// Sequential SDOs at startup or when forced; parallel writes otherwise (mirrors Homing Params block).
FUNCTION_BLOCK FB_WriteStepModeParameters
VAR_INPUT
    bEnable : BOOL;
END_VAR
VAR_IN_OUT
    stDS402Drive         : ST_DS402Drive;
    stMotionStage        : ST_MotionStage;
    stMCS2ChanParameter	: ST_MCS2ChanParameter;
END_VAR

VAR_OUTPUT
   bStepModeParamsSet : BOOL;
END_VAR
VAR
    // ====== Measurements & scaled values ======
    {attribute 'hide'}
    nScaledFErrWin          : DINT;
    {attribute 'hide'}
    nScalededSteps          : DINT;
    {attribute 'hide'}
    fScalededSteps          : LREAL;
    {attribute 'hide'}
    fMeasuredVelo           : LREAL;
    {attribute 'hide'}
    fMeasuredAcc            : LREAL;
    {attribute 'hide'}
    fParameterValue         : LREAL;
    {attribute 'hide'}
    fMeasuredPos             : LREAL;
    // ====== Internal numeric parameters ======
    {attribute 'hide'}
    nScalededStepAmp         : UINT;
    {attribute 'hide'}
    nScaledStepFreq          : UINT;
    // Open Loop Operations
    {attribute 'hide'}
    fbSetSteps          : FB_EcCoESdoWrite;
    {attribute 'hide'}
    fbSetStepFreq       : FB_EcCoESdoWrite;
    {attribute 'hide'}
    fbSetStepAmp        : FB_EcCoESdoWrite;
    {attribute 'hide'}
    nRecentSteps        : DINT;
    {attribute 'hide'}
    nRecentStepAmp      : UINT;
    {attribute 'hide'}
    nRecentStepFreq     : UINT;
    {attribute 'hide'}
    ftStepAmpUpdateDone : F_TRIG;
    {attribute 'hide'}
    ftStepFreqUpdateDone    : F_TRIG;
    {attribute 'hide'}
    ftStepUpdateDone    : F_TRIG;
    tonStartUp : TON;
    nJogParamStep : INT := 0; // 0=idle/start, 1=steps, 2=amp, 3=freq, 10=done, -1=error
    bForceSequentialSDOs : BOOL := FALSE;
    bErrorAcknowledge: BOOL;
END_VAR

IF bEnable THEN
    tonStartUp(
        IN := bEnable AND NOT bStepModeParamsSet,
        PT := T#4S
    );
    IF (NOT tonStartUp.Q) AND (nJogParamStep <> 0) AND (NOT bForceSequentialSDOs) THEN
        nJogParamStep := 0;
    END_IF

    IF (nJogParamStep = -1) AND bErrorAcknowledge THEN
        nJogParamStep := 0;
        stMotionStage.bError := FALSE;
        stMotionStage.nErrorId := 0;
    END_IF
    ScaleStepModeParams();

    ftStepUpdateDone   (CLK := fbSetSteps.bBusy);
    ftStepAmpUpdateDone(CLK := fbSetStepAmp.bBusy);
    ftStepFreqUpdateDone(CLK := fbSetStepFreq.bBusy);

    IF tonStartUp.Q OR bForceSequentialSDOs THEN
        CASE nJogParamStep OF
        0:
            bStepModeParamsSet := FALSE;
            fbSetSteps.bExecute     := FALSE;
            fbSetStepAmp.bExecute   := FALSE;
            fbSetStepFreq.bExecute  := FALSE;
            nJogParamStep := 1;

        1: // Set Steps
            IF (nScalededSteps <> nRecentSteps) THEN
                fbSetSteps.bExecute := TRUE;
                IF ftStepUpdateDone.Q THEN
                    IF fbSetSteps.bError THEN
                        stMotionStage.bError := fbSetSteps.bError;
                        stMotionStage.nErrorId := fbSetSteps.nErrId;
                        nJogParamStep := -1;
                    ELSE
                        nRecentSteps := nScalededSteps;
                        fbSetSteps.bExecute := FALSE;
                        nJogParamStep := 2;
                    END_IF
                END_IF
            ELSE
                nJogParamStep := 2;
            END_IF

        2: // Set Step Amp
            IF (nScalededStepAmp <> nRecentStepAmp) THEN
                fbSetStepAmp.bExecute := TRUE;
                IF ftStepAmpUpdateDone.Q THEN
                    IF fbSetStepAmp.bError THEN
                        stMotionStage.bError := fbSetStepAmp.bError;
                        stMotionStage.nErrorId := fbSetStepAmp.nErrId;
                        nJogParamStep := -1;
                    ELSE
                        nRecentStepAmp := nScalededStepAmp;
                        fbSetStepAmp.bExecute := FALSE;
                        nJogParamStep := 3;
                    END_IF
                END_IF
            ELSE
                nJogParamStep := 3;
            END_IF

        3: // Set Step Frequency
            IF (nScaledStepFreq <> nRecentStepFreq) THEN
                fbSetStepFreq.bExecute := TRUE;
                IF ftStepFreqUpdateDone.Q THEN
                    IF fbSetStepFreq.bError THEN
                        stMotionStage.bError := fbSetStepFreq.bError;
                        stMotionStage.nErrorId := fbSetStepFreq.nErrId;
                        nJogParamStep := -1;
                    ELSE
                        nRecentStepFreq := nScaledStepFreq;
                        fbSetStepFreq.bExecute := FALSE;
                        nJogParamStep := 10;
                    END_IF
                END_IF
            ELSE
                nJogParamStep := 10;
            END_IF

        10: // Done
            bStepModeParamsSet := TRUE;
        -1: // Error state
            bStepModeParamsSet := FALSE;
        ELSE
            nJogParamStep := 0;
        END_CASE

    ELSE
        fbSetSteps.bExecute    := (nScalededSteps   <> nRecentSteps);
        fbSetStepAmp.bExecute  := (nScalededStepAmp <> nRecentStepAmp);
        fbSetStepFreq.bExecute := (nScaledStepFreq  <> nRecentStepFreq);

        IF ftStepUpdateDone.Q OR ftStepAmpUpdateDone.Q OR ftStepFreqUpdateDone.Q THEN
            IF fbSetSteps.bError THEN
                stMotionStage.bError := fbSetSteps.bError;
                stMotionStage.nErrorId := fbSetSteps.nErrId;
            ELSIF fbSetStepAmp.bError THEN
                stMotionStage.bError := fbSetStepAmp.bError;
                stMotionStage.nErrorId := fbSetStepAmp.nErrId;
            ELSIF fbSetStepFreq.bError THEN
                stMotionStage.bError := fbSetStepFreq.bError;
                stMotionStage.nErrorId := fbSetStepFreq.nErrId;
            ELSE
                nRecentSteps    := nScalededSteps;
                nRecentStepAmp  := nScalededStepAmp;
                nRecentStepFreq := nScaledStepFreq;
                bStepModeParamsSet := TRUE;
            END_IF

            fbSetSteps.bExecute    := FALSE;
            fbSetStepAmp.bExecute  := FALSE;
            fbSetStepFreq.bExecute := FALSE;
        END_IF
    END_IF

    fbSetSteps(
        sNetId     := stMotionStage.stAxisParameters.sAmsNetId,
        nSlaveAddr := stDS402Drive.nSlaveAddr,
        nIndex     := stMCS2ChanParameter.nChanStepIdx,
        nSubIndex  := 0,
        pSrcBuf    := ADR(nScalededSteps),
        cbBufLen   := SIZEOF(stMCS2ChanParameter.nChanStep)
    );
    fbSetStepAmp(
        sNetId     := stMotionStage.stAxisParameters.sAmsNetId,
        nSlaveAddr := stDS402Drive.nSlaveAddr,
        nIndex     := stMCS2ChanParameter.nChanStepAmpIdx,
        nSubIndex  := 0,
        pSrcBuf    := ADR(nScalededStepAmp),
        cbBufLen   := SIZEOF(stMCS2ChanParameter.nChanStepAmp)
    );
    fbSetStepFreq(
        sNetId     := stMotionStage.stAxisParameters.sAmsNetId,
        nSlaveAddr := stDS402Drive.nSlaveAddr,
        nIndex     := stMCS2ChanParameter.nChanStepFreqIdx,
        nSubIndex  := 0,
        pSrcBuf    := ADR(nScaledStepFreq),
        cbBufLen   := SIZEOF(stMCS2ChanParameter.nChanStepFreq)
    );

    bStepModeParamsSet R= fbSetSteps.bBusy
        OR fbSetStepAmp.bBusy
        OR fbSetStepFreq.bBusy;
END_IF

(*Scaled Open Loop Step mode motion parameters*)
METHOD ScaleStepModeParams
VAR_INPUT
END_VAR
//827.31x-837.63
nScalededSteps:=LIMIT(-1000, stMCS2ChanParameter.nChanStep, 1000);
nScalededStepAmp:=REAL_TO_UINT(LIMIT(50, stMCS2ChanParameter.nChanStepAmp, 100) * 655.35);
nScaledStepFreq:=REAL_TO_UINT(LIMIT(500, stMCS2ChanParameter.nChanStepFreq, 1000.0));
END_METHOD

END_FUNCTION_BLOCK

(* stored: Version 1.1.0.1
   POU FB_WriteStepModeParameters: Id {309453e5-6198-4e60-a7a5-fef2f5a9da17}, SpecialFunc None
   Method ScaleStepModeParams: Id {78ce5a79-ef3b-44af-a794-7ac04154475b} *)
